FUNCTION_BLOCK SledgeHAL
  (* Standard: 61499-2 *)
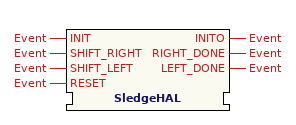
  EVENT_INPUT
    INIT;
    SHIFT_RIGHT;
    SHIFT_LEFT;
    RESET;
  END_EVENT
  EVENT_OUTPUT
    INITO;
    RIGHT_DONE;
    LEFT_DONE;
  END_EVENT
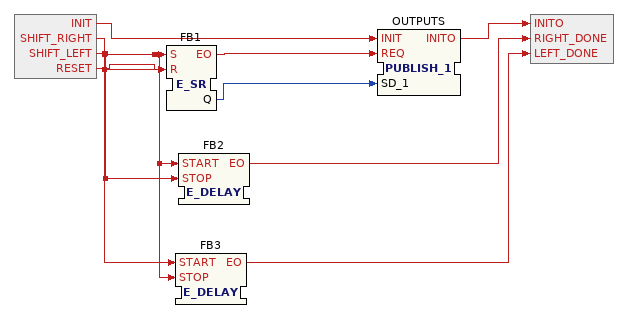
  FBS
    OUTPUTS : PUBLISH_1;
    FB1 : E_SR;
    FB2 : E_DELAY;
    FB3 : E_DELAY;
  END_FBS
  EVENT_CONNECTIONS
    INIT TO OUTPUTS.INIT;
    OUTPUTS.INITO TO INITO;
    SHIFT_RIGHT TO FB1.S;
    SHIFT_LEFT TO FB1.R;
    FB1.EO TO OUTPUTS.REQ;
    FB2.EO TO RIGHT_DONE;
    FB3.EO TO LEFT_DONE;
    SHIFT_RIGHT TO FB2.START;
    SHIFT_LEFT TO FB2.STOP;
    SHIFT_LEFT TO FB3.START;
    SHIFT_RIGHT TO FB3.STOP;
    RESET TO FB1.R;
  END_CONNECTIONS
  DATA_CONNECTIONS
    FB1.Q TO OUTPUTS.SD_1;
  END_CONNECTIONS
END_FUNCTION_BLOCK
